(* PLC project Blank Project, Blank Blank 1.0 *)
(* stored: creationDateTime 2016-05-18T21:14:07, modificationDateTime 2016-11-21T18:27:12 *)

PROGRAM Cell3
  VAR
    C2_IR AT %IX0.3 : BOOL := true;
    M2_IR AT %IX0.4 : BOOL := true;
    Main AT %IX0.6 : BOOL := true;
    M2_motor AT %QX0.2 : BOOL := true;
    C3_motor AT %QX0.4 : BOOL := true;
  END_VAR
  VAR
    C3_working : BOOL := false;
  END_VAR
  VAR
    C3_working_int AT %MD1 : DINT := 0;
  END_VAR
  VAR
    M2_working : BOOL := false;
  END_VAR
  VAR
    M2_working_int AT %MD3 : DINT := 0;
  END_VAR
  VAR
    Timer_conveyor : TON;
    Timer_machining : TON;
  END_VAR

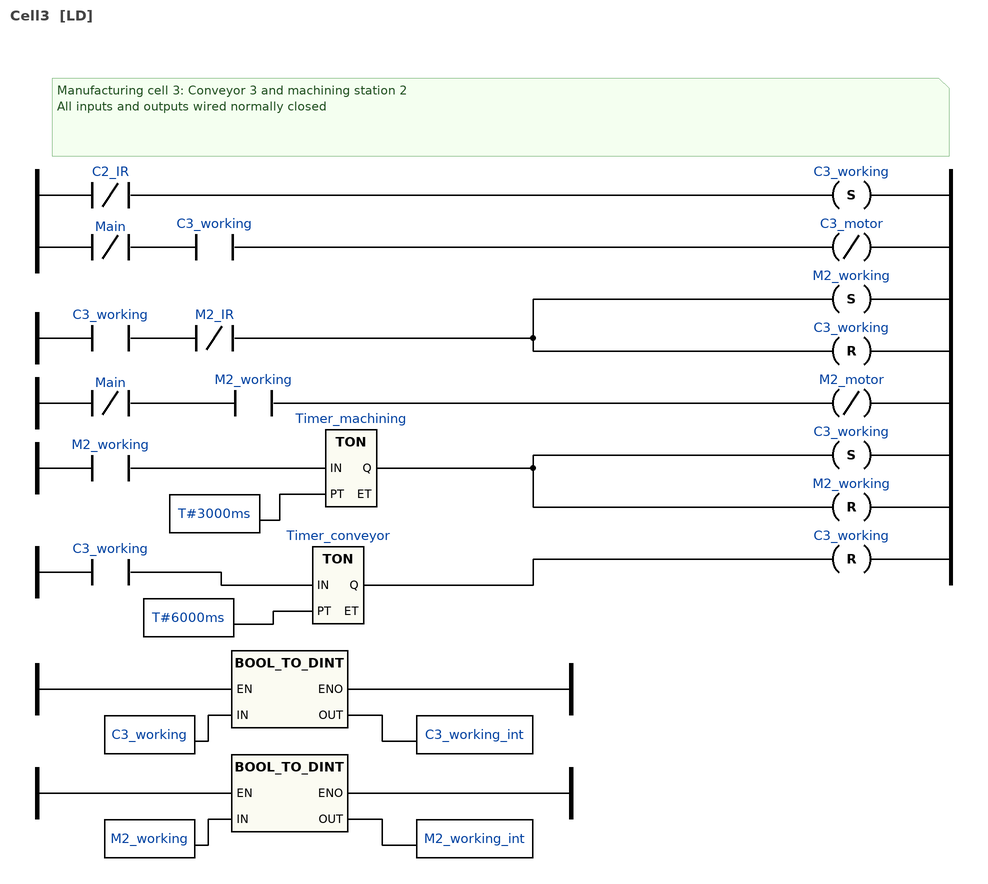
(* LD diagram, written out as Structured Text *)
(* Manufacturing cell 3: Conveyor 3 and machining station 2
All inputs and outputs wired normally closed *)
IF NOT C2_IR THEN C3_working := TRUE; END_IF;
C3_motor := NOT (NOT Main AND C3_working);
IF C3_working AND NOT M2_IR THEN M2_working := TRUE; END_IF;
IF C3_working AND NOT M2_IR THEN C3_working := FALSE; END_IF;
M2_motor := NOT (NOT Main AND M2_working);
Timer_machining(IN := M2_working, PT := T#3000ms);
IF Timer_machining.Q THEN C3_working := TRUE; END_IF;
IF Timer_machining.Q THEN M2_working := FALSE; END_IF;
Timer_conveyor(IN := C3_working, PT := T#6000ms);
IF Timer_conveyor.Q THEN C3_working := FALSE; END_IF;
C3_working_int := BOOL_TO_DINT(C3_working);
M2_working_int := BOOL_TO_DINT(M2_working);
END_PROGRAM

CONFIGURATION Config0
  RESOURCE Res0 ON PLC
    TASK TaskMain(INTERVAL := T#50ms, PRIORITY := 0);
    PROGRAM Inst0 WITH TaskMain : Cell3;
  END_RESOURCE
END_CONFIGURATION
